// TIA Portal V18 export
TYPE "UDT_MES_UnLoadData_ext"
// stored: IsFailsafeCompliant false
   STRUCT
      "PLC.CheckSum" : Int;   // 校验和
      "PLC.PartTypeID" : Int;   // 产品类型
      "PLC.PartTypeSN" : String[50];   // 产品主体码
      "PLC.SubPartSN" : String[50];   // 产品组件码
      "PLC.PartStatus" : DInt;   // 产品加工结果（1 OK;2 NG）
      "PLC.StatusBits2" : DInt;
      "PLC.Result" : Array[1..150] of Real;
      "MES.ErrorCode" : Int;   // 异常代码
      "MES.ErrorMsg" : String[50];   // 异常信息
   END_STRUCT;
END_TYPE
